// Converts internal loglevel to twincat severity
FUNCTION LogLevel_To_Severity : TcEventSeverity
VAR_INPUT
	eLogLevel:				E_LogLevel;
END_VAR
VAR
END_VAR

CASE eLogLevel OF
	E_LogLevel.Verbose:
		LogLevel_To_Severity:= TcEventSeverity.Verbose;
		
	E_LogLevel.Info:
		LogLevel_To_Severity:= TcEventSeverity.Info;
		
	E_LogLevel.Warning:
		LogLevel_To_Severity:= TcEventSeverity.Warning;
		
	E_LogLevel.Error:
		LogLevel_To_Severity:= TcEventSeverity.Error;
		
	E_LogLevel.Critical:
		LogLevel_To_Severity:= TcEventSeverity.Critical;
		
END_CASE

END_FUNCTION

(* stored: Version 1.1.0.1
   POU LogLevel_To_Severity: Id {2125d2a6-85a2-44a9-b27f-c4f068813b29}, SpecialFunc None *)
